// SIMATIC S7-200 SMART project (STEP 7-Micro/WIN SMART), CPU SR40

ORGANIZATION_BLOCK MAIN:OB1
TITLE=Program Comments
BEGIN
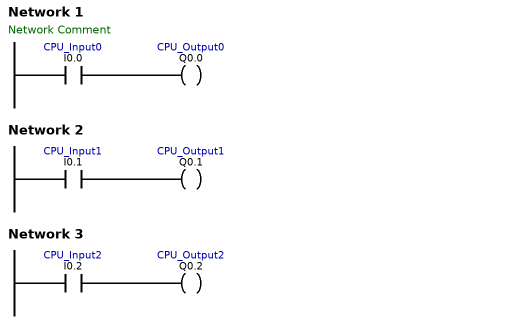
Network 1
// Network Comment
LD     CPU_Input0:I0.0
=      CPU_Output0:Q0.0
Network 2
LD     CPU_Input1:I0.1
=      CPU_Output1:Q0.1
Network 3
LD     CPU_Input2:I0.2
=      CPU_Output2:Q0.2
END_ORGANIZATION_BLOCK
